// TwinCAT 3 PLC project PTP_PLC
// ProgramVersion: 3.1.4022.3
// libraries:
//   Tc2_EtherCAT, * (Beckhoff Automation GmbH)
//   Tc2_Standard, * (Beckhoff Automation GmbH)
//   Tc2_System, * (Beckhoff Automation GmbH)
//   Tc3_Module, * (Beckhoff Automation GmbH)
// project tree:
//   DUTs/ TimeInfo.TcDUT
//   / PlcTask.TcTTO
//   POUs/ MAIN.TcPOU
// real-time tasks:
//   TASK PlcTask: cycle T#1ms, priority 20, ADS port 350
// I/O:
//   DEVICE Device 1 (EtherCAT), AmsNetId 5.56.86.54.2.1
//     Term 1 (EK1200) [EK1200-5000 EtherCAT Power supply (2A E-Bus)]
//       Term 2 (EL1819) [EL1819 16Ch. Dig. Input 24V, 10µs]
//       Term 3 (EL6688) [EL6688 - External Synchronisation Interface (IEEE1588)]
//       Term 4 (EL9011) [EL9011 End Terminal]
// variable links:
//   PTP_PLC/PTP_PLC Instance <-> Device 1 (EtherCAT)
//     PlcTask Inputs/MAIN.dctoextoff <-> InfoData/DcToExtTimeOffset
//     PlcTask Inputs/MAIN.dctotcoff <-> InfoData/DcToTcTimeOffset
//   PTP_PLC/PTP_PLC Instance <-> Device 1 (EtherCAT)/Term 1 (EK1200)/Term 3 (EL6688)
//     PlcTask Inputs/MAIN.externalstamp <-> External Sync/External time stamp
//     PlcTask Inputs/MAIN.internalstamp <-> External Sync/Internal time stamp

CONFIGURATION PTP_PLC
    RESOURCE PLC ON TwinCAT3
        TASK PlcTask(INTERVAL := T#1ms, PRIORITY := 20);
        PROGRAM MAIN WITH PlcTask : MAIN;
    END_RESOURCE
END_CONFIGURATION

// ---- DUTs/TimeInfo.TcDUT
TYPE TimeInfo :
STRUCT
	dctime: T_DCTIME64; (* The DC time gotten from F_GetActualDcTime64(). *)
    dctotcoff: LINT; (* Offset between DC and TwinCAT time (in ns). *)
	dctoextoff: LINT; (* Offset between DC and external time (in ns). *)
	internalstamp: ULINT; (* Internal timestamp from EL6688. *)
	externalstamp: ULINT; (* External timestamp from EL6688. *)
END_STRUCT
END_TYPE

// ---- POUs/MAIN.TcPOU
PROGRAM MAIN
VAR
	dctotcoff AT %I*: LINT; (* Offset between DC and TwinCAT time (in ns). *)
	dctoextoff AT %I*: LINT; (* Offset between DC and external time (in ns). *)
	internalstamp AT %I*: ULINT; (* Internal timestamp from EL6688. *)
	externalstamp AT %I*: ULINT; (* External timestamp from EL6688. *)
	first: BOOL := TRUE;
	timer: TON;
	tinfo: TimeInfo;
END_VAR

IF first THEN
	first := FALSE;
	timer(in:=FALSE, pt:=T#1S);
END_IF
timer(in:=TRUE);
IF timer.Q THEN
	tinfo.dctime := F_GetActualDcTime64();
	tinfo.dctoextoff := dctoextoff;
	tinfo.dctotcoff := dctotcoff;
	tinfo.externalstamp := externalstamp;
	tinfo.internalstamp := internalstamp;
	timer(in:=FALSE);
END_IF

END_PROGRAM
